///////////
// Structure For I35. Main Operating Data to be saved ( ex: OPC ) .  
//////////
TYPE UPS_CXC :
STRUCT
	
	MesData				: UPS ; 	(* Object 									*)
	            		            (*                                          *)
	MesU				: REAL ; 	(*(V) AC voltage                            *)
	MesIload			: REAL ; 	(*(A) DC Load current                       *)
	MesUBatt			: REAL ; 	(*(V) Battery voltage                       *)
	MesIBatt			: REAL ; 	(*(A) Battery Current                       *)
	MesSoC  			: REAL ; 	(*(%) Battery SoC                           *)
	MesIdc  			: REAL ; 	(*(A) battery + load Current                *)

	
	MesOverTempBatt 	: BOOL ; 	(* OverTemperature of the battery alarm		*)
	MesCBUpsOpened		: BOOL ; 	(* UPS CB opened alarm                      *)
	
		
	
END_STRUCT
END_TYPE

(* stored: Version 1.1.0.1, ProductVersion 3.1.4024.6
   DUT UPS_CXC: Id {87df5298-94a3-4d4c-8d7f-664483729d5b} *)
